Fanuc KAREL source: ko00087.KL

PROGRAM KO00087
%STACKSIZE=65535
%PRIORITY=65535
%NOLOCKGROUP
VAR
P1 : JOINTPOS9
P2 : XYZWPR
F : BOOLEAN
OUT : XYZWPREXT
BEGIN
F=TRUE
-- UNSAFE_SOURCE_IR line 11: OUT = MIRROR(convert_jointpos9_to_xyzwprext(P1), convert_xyzwpr_to_position(P2), F)
END KO00087
